Staubli VAL3: socketServer.pjx

--- socketServer.pjx ---
Parameters version=s7.9.1 stackSize=5000 millimeterUnit=true
Program file=actGesture.pgx
Program file=actMovement.pgx
Program file=dataGet.pgx
Program file=detectInput.pgx
Program file=gestureFist.pgx
Program file=parseMovement.pgx
Program file=start.pgx
Program file=stop.pgx
Data file=socketServer.dtx

--- socketServer.dtx ---
mdesc nom_speed = {rmax=9999, blend=off}
sio sioSocket = {link=Socket\HelloServer}
num nNum
num nBuffer
string sBuffer
string sInput[50]
num nFailCounter
jointRx jTest
pointRs pPointRs = {fatherId=world[0]}
bool bDetectInput
tool tClaw = {z=90, fatherId=flange[0], ioLink=valve1}
bool bClawClosed
num nMovementData[3]

--- start.pgx ---
public program start()
begin
  nBuffer = 0
  nNum = 0
  nFailCounter = 0
  bDetectInput = false
  sInput = ""
  //call enablePowerTest()
  call detectInput()
end

--- actGesture.pgx ---
program actGesture()
begin
  putln("GestureCalled")
  putln(sInput)
  if (sInput == "fist")
    call gestureFist()
  endIf

end

--- actMovement.pgx ---
program actMovement()
begin
  putln("actMovement called")
  putln(sInput)

end

--- dataGet.pgx ---
program dataGet()
begin
  //dataGet essentially gathers all of the inputs together and then calls the appropiate method
  //It is VITAL that the signal sent ends in either a ) (gesture) and } (movement).
  sBuffer = chr(nBuffer)
  putln(sBuffer)
  if(sBuffer == ")")
    //putln("dataGet")
    call actGesture()
    sInput = ""
    nBuffer = 0
    sBuffer = ""
  elseIf(sBuffer == "}")
    //putln(sInput)
    call parseMovement()
    //sInput = ""
  else
    sInput = sInput + sBuffer
  endIf
  //sBuffer = ""
end

--- detectInput.pgx ---
program detectInput()
begin
  //Detect input detects if it is getting a signal and then calls the dataGet
  //method. Which creates the input. Since if I sent "hellWorld" through the client to the server. It would
  //be sent one character at a time. That is why we have the while loop. sioGet has a very useful function where it will
  //pause the entire program until it recieves a signal. Preventing the while loop from iterating.
  while true
    nNum = sioGet(sioSocket,nBuffer)
    putln(nNum)
    if nNum >= 0
      if nBuffer != 0
        putln("dataGet called")
        call dataGet()
      endIf
    endIf
  endWhile
end

--- gestureFist.pgx ---
program gestureFist()
begin
    if (bClawClosed == false)
      close(tClaw)
      putln("Fist Closed")
      bClawClosed = true
    elseIf (bClawClosed == true)
      open(tClaw)
      putln("Fist Opened")
      bClawClosed = false
    endIf
end

--- parseMovement.pgx ---
program parseMovement()
begin
  putln(sInput)
end

--- stop.pgx ---
program stop()
begin
  popUpMsg("Pending movement commands have been canceled")
  resetMotion()
end
